// TIA Portal V19 export
TYPE "LEXCHANGETRAY_typeConstraintWorkstation_signalTM_ControlNode"
// stored: Access Published
   STRUCT
      cmd : "LEXCHANGETRAY_typeConstraintWorkstation_signalTM_Cmd";
      monitor { S7_SetPoint := 'True'} : "LEXCHANGETRAY_typeConstraintWorkstation_signalTM_Monitor";
      sim { S7_SetPoint := 'True'} : "LEXCHANGETRAY_typeConstraintWorkstation_signalTM_Simulation";
   END_STRUCT;
END_TYPE
